SUBAPPLICATION Zaehler (* Subapplication Type *)
  (* Standard: 61499-2 *)
  (* Version 1.0, 2023-02-17, Franz *)
  PACKAGE FBs::Counter::subs::Zaehler;
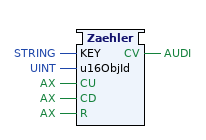
  VAR_INPUT
    KEY : STRING;
    u16ObjId : UINT;
  END_VAR
  SOCKETS
    CU : adapter::types::unidirectional::AX; (* Count Up *)
    CD : adapter::types::unidirectional::AX; (* Count Down *)
    R : adapter::types::unidirectional::AX; (* Reset *)
  END_SOCKETS
  PLUGS
    CV : adapter::types::unidirectional::AUDI; (* Counter Value *)
  END_PLUGS
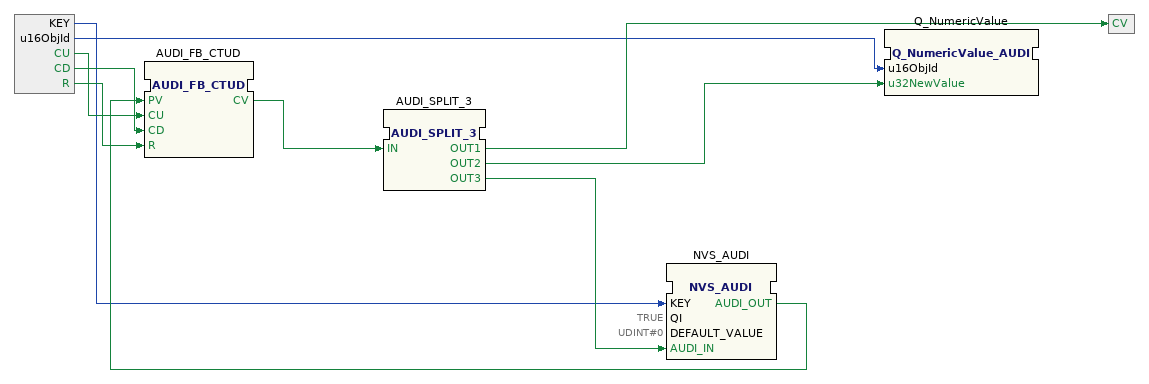
  FBS
    AUDI_FB_CTUD : adapter::iec61131::counters::AUDI_FB_CTUD;
    Q_NumericValue : isobus::UT::Q::Q_NumericValue_AUDI;
    NVS_AUDI : logiBUS::storage::esp32_nvs::NVS_AUDI(QI := TRUE, DEFAULT_VALUE := UDINT#0);
    AUDI_SPLIT_3 : adapter::events::unidirectional::AUDI_SPLIT_3;
  END_FBS
  DATA_CONNECTIONS
    u16ObjId TO Q_NumericValue.u16ObjId;
    KEY TO NVS_AUDI.KEY;
  END_CONNECTIONS
  ADAPTER_CONNECTIONS
    AUDI_FB_CTUD.CV TO AUDI_SPLIT_3.IN;
    NVS_AUDI.AUDI_OUT TO AUDI_FB_CTUD.PV;
    AUDI_SPLIT_3.OUT1 TO CV;
    AUDI_SPLIT_3.OUT2 TO Q_NumericValue.u32NewValue;
    AUDI_SPLIT_3.OUT3 TO NVS_AUDI.AUDI_IN;
    CU TO AUDI_FB_CTUD.CU;
    CD TO AUDI_FB_CTUD.CD;
    R TO AUDI_FB_CTUD.R;
  END_CONNECTIONS
END_SUBAPPLICATION
